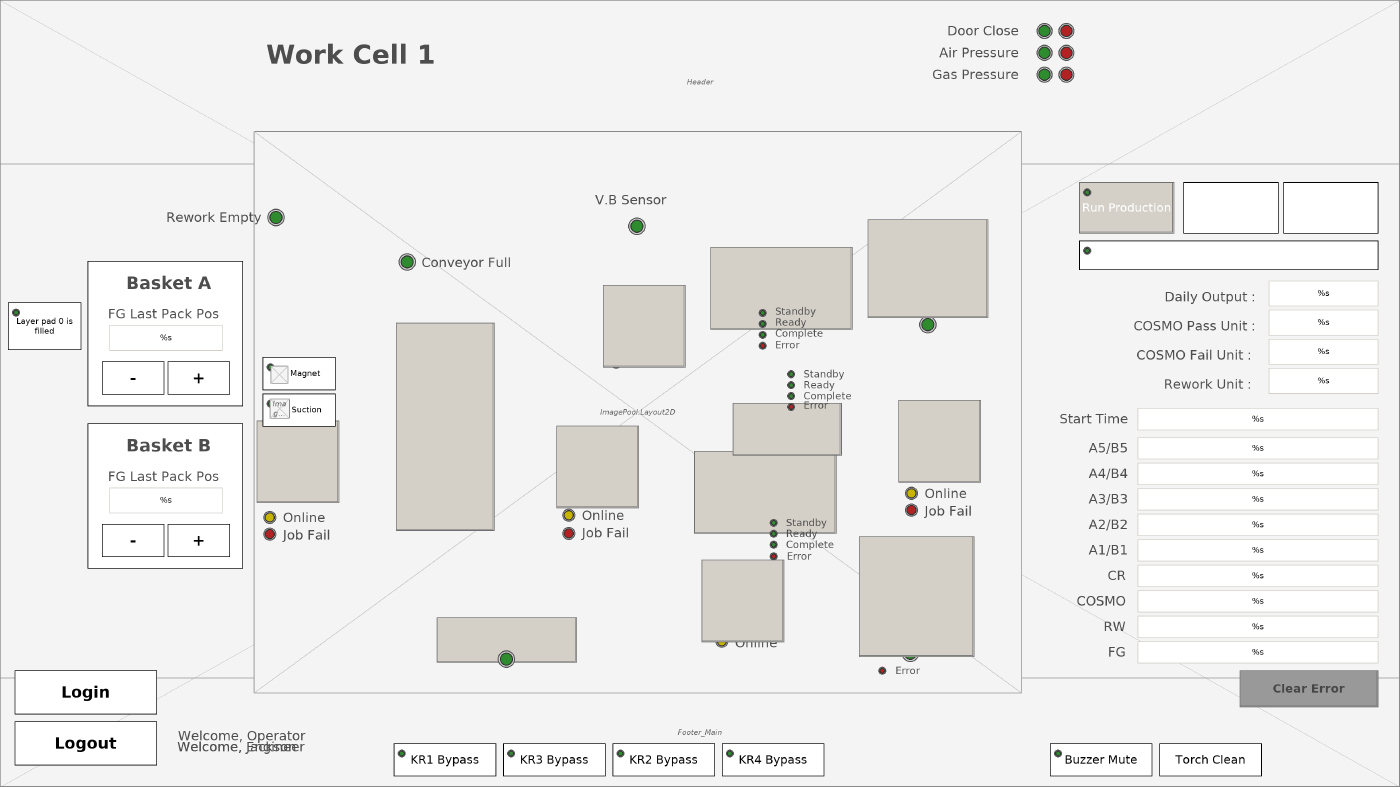
VISUALIZATION PAGE_MAIN  // 1920x1080
    Image (0,0 1920x1080), image: ImagePool.The-New-Silver-Backgrounds
    Frame (0,930 1920x150)
        shows Footer_Main()
        shows Footer_1()
    Frame (0,0 1920x225)
        shows Header()
    Label (362,45 650x60), "Work Cell 1"
    RoundedRectangle (1760,250 130x70), "Reset Production"
        OnMouseClick: OpenDialog Dialog=MSG_BOX_RESET, OpenModal=True, OpenCentered=True
    RoundedRectangle (20,990 195x60), "Logout"
        OnMouseClick: VisuUserMgmt Type=Logout
        OnMouseClick: execute {
            LOGFILE( sLogEvent	 := MSG.EVENT_BTN,
            		 sLogComp	 := MSG.COMP_HMI,
            		 sLogAction	 := MSG.ACTION_LOGOUT,
            	 	 logFlag	 := TRUE);
        }
    RoundedRectangle (20,920 195x60), "Login"
        tap MAIN.BTN_LOG
        OnMouseClick: VisuUserMgmt Type=Login
        OnMouseClick: execute {
            LOGFILE( sLogEvent	 := MSG.EVENT_BTN,
            		 sLogComp	 := MSG.COMP_HMI,
            		 sLogAction	 := MSG.ACTION_LOGIN,
            	 	 logFlag	 := TRUE);
        }
    Label (240,1005 200x40), "Welcome, Engineer"
    Label (240,1005 200x40), "Welcome, Jackson"
    Label (241,990 200x40), "Welcome, Operator"
    RoundedRectangle (120,358 213x199)
    Label (170,366 119x45), "Basket A"
    RoundedRectangle (140,496 85x45), "-"
        tap JIG.BasketA_Minus
        OnMouseClick: execute {
            LOGFILE( sLogEvent	 := MSG.EVENT_BTN,
            		 sLogComp	 := MSG.COMP_FG,
            		 sLogAction	 := MSG.ACTION_BSKTA_MINUS,
            	 	 logFlag	 := TRUE);
        }
    RoundedRectangle (230,496 85x45), "+"
        tap JIG.BasketA_Plus
        OnMouseClick: execute {
            LOGFILE( sLogEvent	 := MSG.EVENT_BTN,
            		 sLogComp	 := MSG.COMP_FG,
            		 sLogAction	 := MSG.ACTION_BSKTA_PLUS,
            	 	 logFlag	 := TRUE);
        }
    Textfield (150,446 155x35), "%s", text variable: GVL.Basket_A_Counter
    Label (145,416 173x30), "FG Last Pack Pos"
    RoundedRectangle (120,581 213x199)
    Label (170,589 119x45), "Basket B"
    RoundedRectangle (140,719 85x45), "-"
        tap JIG.BasketB_Minus
        OnMouseClick: execute {
            LOGFILE( sLogEvent	 := MSG.EVENT_BTN,
            		 sLogComp	 := MSG.COMP_FG,
            		 sLogAction	 := MSG.ACTION_BSKTA_MINUS,
            	 	 logFlag	 := TRUE);
        }
    RoundedRectangle (230,719 85x45), "+"
        tap JIG.BasketB_Plus
        OnMouseClick: execute {
            LOGFILE( sLogEvent	 := MSG.EVENT_BTN,
            		 sLogComp	 := MSG.COMP_FG,
            		 sLogAction	 := MSG.ACTION_BSKTB_PLUS,
            	 	 logFlag	 := TRUE);
        }
    Textfield (150,669 155x35), "%s", text variable: GVL.Basket_B_Counter
    Label (145,639 173x30), "FG Last Pack Pos"
    Image (348,180 1053x771), image: ImagePool.Layout2D
    Lamp1 (865,430 27x27), variable: KR3.bInBit[1,6], style: Lamp-Lamp1-Green
    Lamp1 (1010,815 27x27), variable: KR4.bInBit[1,6], style: Lamp-Lamp1-Green
    Lamp1 (1275,600 27x27), variable: KR5.bInBit[1,6], style: Lamp-Lamp1-Green
    Lamp1 (800,625 27x27), variable: KR2.bInBit[1,6], style: Lamp-Lamp1-Green
    Lamp1 (360,700 20x20), variable: KR1.KROnline, style: Lamp-Lamp1-Yellow
    Button (543,443 135x285)
        OnMouseClick: change screen: PAGE_CoolRack
        OnMouseClick: execute {
            LOGFILE( sLogEvent	 := MSG.EVENT_PAGE,
            		 sLogComp	 := MSG.COMP_CR,
            		 sLogAction	 := MSG.ACTION_COOLRACK,
            	 	 logFlag	 := TRUE);
        }
    Button (599,847 192x62)
        OnMouseClick: change screen: PAGE_COSMO
        OnMouseClick: execute {
            LOGFILE( sLogEvent	 := MSG.EVENT_PAGE,
            		 sLogComp	 := MSG.COMP_CM,
            		 sLogAction	 := MSG.ACTION_COSMO,
            	 	 logFlag	 := TRUE);
        }
    Lamp1 (681,891 27x27), variable: GVL.COSMO_Ready, style: Lamp-Lamp1-Green
    Lamp1 (860,297 27x27), variable: GVL.VibBowl_Ready, style: Lamp-Lamp1-Green
    Label (813,252 255x45), "V.B Sensor"
    Lamp1 (1259,432 27x27), variable: INFEED_RACK.IFRack_Ready, style: Lamp-Lamp1-Green
    Lamp1 (1235,883 27x27), variable: GVL.JIGC_Standby, style: Lamp-Lamp1-Green
    Button (1178,736 158x165)
        OnMouseClick: change screen: PAGE_TTorch
        OnMouseClick: execute {
            LOGFILE( sLogEvent	 := MSG.EVENT_PAGE,
            		 sLogComp	 := MSG.COMP_TT,
            		 sLogAction	 := MSG.ACTION_TT,
            	 	 logFlag	 := TRUE);
        }
    Button (974,339 195x113)
        OnMouseClick: change screen: PAGE_JIG_A
        OnMouseClick: execute {
            LOGFILE( sLogEvent	 := MSG.EVENT_PAGE,
            		 sLogComp	 := MSG.COMP_JIGA,
            		 sLogAction	 := MSG.ACTION_JIGA,
            	 	 logFlag	 := TRUE);
        }
    Button (952,619 195x113)
        OnMouseClick: change screen: PAGE_JIG_C
        OnMouseClick: execute {
            LOGFILE( sLogEvent	 := MSG.EVENT_PAGE,
            		 sLogComp	 := MSG.COMP_JIGC,
            		 sLogAction	 := MSG.ACTION_JIGC,
            	 	 logFlag	 := TRUE);
        }
    Button (1005,553 149x72)
        OnMouseClick: change screen: PAGE_JIG_B
        OnMouseClick: execute {
            LOGFILE( sLogEvent	 := MSG.EVENT_PAGE,
            		 sLogComp	 := MSG.COMP_JIGB,
            		 sLogAction	 := MSG.ACTION_JIGB,
            	 	 logFlag	 := TRUE);
        }
    Lamp1 (365,285 27x27), variable: GVL.Rework_Empty, style: Lamp-Lamp1-Green
    Lamp1 (545,346 27x27), variable: GVL.Conveyor_Full, style: Lamp-Lamp1-Green
    Label (225,276 146x45), "Rework Empty"
    Label (575,338 130x45), "Conveyor Full"
    Lamp1 (360,723 20x20), variable: KR1.bInBit[4,0], style: Lamp-Lamp1-Red
    Lamp1 (1240,690 20x20), variable: KR5.bInBit[4,7], style: Lamp-Lamp1-Red
    Lamp1 (770,722 20x20), variable: KR2.bInBit[3,4], style: Lamp-Lamp1-Red
    Lamp1 (395,633 27x27), variable: KR1.bInBit[1,6], style: Lamp-Lamp1-Green
    Label (385,722 80x25), "Job Fail"
    Label (385,698 80x25), "Online"
    Lamp1 (770,697 20x20), variable: KR2.KROnline, style: Lamp-Lamp1-Yellow
    Label (795,719 80x25), "Job Fail"
    Label (795,695 80x25), "Online"
    Lamp1 (1240,667 20x20), variable: KR5.KROnline, style: Lamp-Lamp1-Yellow
    Label (1265,689 80x25), "Job Fail"
    Label (1265,665 80x25), "Online"
    Lamp1 (835,487 20x20), variable: KR3.KROnline, style: Lamp-Lamp1-Yellow
    Label (860,485 80x25), "Online"
    Lamp1 (980,870 20x20), variable: KR4.KROnline, style: Lamp-Lamp1-Yellow
    Label (1005,870 80x25), "Online"
    Button (827,391 113x113)
        OnMouseClick: change screen: PAGE_KR3
        OnMouseClick: execute {
            LOGFILE( sLogEvent	 := MSG.EVENT_PAGE,
            		 sLogComp	 := MSG.COMP_KR3,
            		 sLogAction	 := MSG.ACTION_KR3,
            	 	 logFlag	 := TRUE);
        }
    Button (763,584 113x113)
        OnMouseClick: change screen: PAGE_KR2
        OnMouseClick: execute {
            LOGFILE( sLogEvent	 := MSG.EVENT_PAGE,
            		 sLogComp	 := MSG.COMP_KR2,
            		 sLogAction	 := MSG.ACTION_KR2,
            	 	 logFlag	 := TRUE);
        }
    Button (962,768 113x113)
        OnMouseClick: change screen: PAGE_KR4
        OnMouseClick: execute {
            LOGFILE( sLogEvent	 := MSG.EVENT_PAGE,
            		 sLogComp	 := MSG.COMP_KR4,
            		 sLogAction	 := MSG.ACTION_KR4,
            	 	 logFlag	 := TRUE);
        }
    Button (1232,549 113x113)
        OnMouseClick: change screen: PAGE_KR5
        OnMouseClick: execute {
            LOGFILE( sLogEvent	 := MSG.EVENT_PAGE,
            		 sLogComp	 := MSG.COMP_KR5,
            		 sLogAction	 := MSG.ACTION_KR5,
            	 	 logFlag	 := TRUE);
        }
    Button (352,577 113x113)
        OnMouseClick: change screen: PAGE_KR1_Tab
        OnMouseClick: execute {
            LOGFILE( sLogEvent	 := MSG.EVENT_PAGE,
            		 sLogComp	 := MSG.COMP_KR1,
            		 sLogAction	 := MSG.ACTION_KR1,
            	 	 logFlag	 := TRUE);
        }
    Label (1500,425 225x45), "COSMO Pass Unit :"
    Textfield (1740,425 150x35), "%s", text variable: GVL.Pass_Counter
    Textfield (1740,465 150x35), "%s", text variable: GVL.Fail_Counter
    Label (1500,465 225x45), "COSMO Fail Unit :"
    Textfield (1560,880 330x30), "%s", text variable: AUTO_MODE.processnameFG
    Group (1430,705 460x30)
        Textfield (130,0 330x30), "%s", text variable: AUTO_MODE.processnameA2
        Label (0,0 120x30), "A2/B2"
    Group (1430,740 460x30)
        Textfield (130,0 330x30), "%s", text variable: AUTO_MODE.processnameA1
        Label (0,0 120x30), "A1/B1"
    Textfield (1560,600 330x30), "%s", text variable: AUTO_MODE.processnameA5
    Label (1430,600 120x30), "A5/B5"
    Group (1430,635 460x30)
        Textfield (130,0 330x30), "%s", text variable: AUTO_MODE.processnameA4
        Label (0,0 120x30), "A4/B4"
    Group (1430,670 460x30)
        Textfield (130,0 330x30), "%s", text variable: AUTO_MODE.processnameA3
        Label (0,0 120x30), "A3/B3"
    Label (1472,880 75x30), "FG"
    Group (1472,845 418x30)
        Textfield (88,0 330x30), "%s", text variable: AUTO_MODE.processnameRW
        Label (0,0 75x30), "RW"
    Group (1472,775 418x30)
        Textfield (88,0 330x30), "%s", text variable: AUTO_MODE.processnameCR
        Label (0,0 75x30), "CR"
    Group (1455,810 435x30)
        Textfield (105,0 330x30), "%s", text variable: AUTO_MODE.processnameCOSMO
        Label (0,0 92x30), "COSMO"
    Lamp1 (1260,358 20x20), variable: INFEED_RACK.IFRack_Ready, style: Lamp-Lamp1-Yellow
    Button (1190,301 165x135)
        OnMouseClick: change screen: PAGE_InfeedRack
        OnMouseClick: execute {
            LOGFILE( sLogEvent	 := MSG.EVENT_PAGE,
            		 sLogComp	 := MSG.COMP_IR,
            		 sLogAction	 := MSG.ACTION_INFEEDRACK,
            	 	 logFlag	 := TRUE);
        }
    Label (1500,385 225x45), "Daily Output :"
    Textfield (1740,385 150x35), "%s", text variable: GVL.daily_output
    Label (1500,505 225x45), "Rework Unit :"
    Textfield (1740,505 150x35), "%s", text variable: GVL.Rework_Counter
    RoundedRectangle (1480,330 410x40), "Welding Mode"
        toggle SAFETY_SENSOR.WELDING_MODE
        OnMouseClick: execute {  }
    RoundedRectangle (1623,250 130x70), "Halt Production", input disabled if: MAIN.btnTorchClean
        OnMouseClick: execute {
            KR1.bOutBit[1,0]:= FALSE;
            KR2.bOutBit[1,0]:= FALSE;
            KR3.bOutBit[1,0]:= FALSE;
            KR4.bOutBit[1,0]:= FALSE;
            KR5.bOutBit[1,0]:= FALSE;
            LOGFILE( sLogEvent	 := MSG.EVENT_BTN,
            		 sLogComp	 := MSG.COMP_HMI,
            		 sLogAction	 := MSG.ACTION_STOP,
            	 	 logFlag	 := TRUE);
            AUTO_MODE.Halt_Production := TRUE;
            AUTO_MODE.AutoMode := False;
        }
    Button (1480,250 130x70), "Run Production", pressed state: AUTO_MODE.AutoMode, input disabled if: MAIN.btnTorchClean
        toggle AUTO_MODE.AutoMode
        OnMouseClick: execute {
            LOGFILE( sLogEvent	 := MSG.EVENT_BTN,
            		 sLogComp	 := MSG.COMP_HMI,
            		 sLogAction	 := MSG.ACTION_START,
            	 	 logFlag	 := TRUE);
            IF AUTO_MODE.AutoMode THEN
            	AUTO_MODE.Start_time := MAIN.fb_TimeStamp.SystemTime;
            END_IF
        }
    Lamp1 (1485,255 12x18), variable: AUTO_MODE.AutoMode, style: Lamp-Lamp1-Green
    Textfield (1560,560 330x30), "%s", text variable: AUTO_MODE.Start_time
    Label (1430,560 120x30), "Start Time"
    Lamp1 (1485,335 12x18), variable: SAFETY_SENSOR.WELDING_MODE, style: Lamp-Lamp1-Green
    Group (1250,20 225x105)
        Group (0,0 225x45)
            Label (0,0 150x45), "Door Close"
            Lamp1 (170,10 25x25), variable: SAFETY_SENSOR.SENSOR_SAFETY_DOOR_CLOSE, style: Lamp-Lamp1-Green
            Lamp1 (200,10 25x25), variable: not SAFETY_SENSOR.SENSOR_SAFETY_DOOR_CLOSE, style: Lamp-Lamp1-Red
        Label (0,30 150x45), "Air Pressure"
        Lamp1 (170,40 25x25), variable: SAFETY_SENSOR.SENSOR_AIR_PRESSURE_OK, style: Lamp-Lamp1-Green
        Lamp1 (200,40 25x25), variable: not SAFETY_SENSOR.SENSOR_AIR_PRESSURE_OK or SAFETY_SENSOR.SENSOR_AIR_PRESSURE_HIGH, style: Lamp-Lamp1-Red
        Label (0,60 150x45), "Gas Pressure"
        Lamp1 (170,70 25x25), variable: SAFETY_SENSOR.SENSOR_GAS_PRESSURE_OK, style: Lamp-Lamp1-Green
        Lamp1 (200,70 25x25), variable: not SAFETY_SENSOR.SENSOR_GAS_PRESSURE_OK or SAFETY_SENSOR.SENSOR_GAS_PRESSURE_HIGH, style: Lamp-Lamp1-Red
    Group (1079,506 100x45)
        Lamp1 (0,0 12x15), variable: GVL.JIGB_Standby, style: Lamp-Lamp1-Green
        Lamp1 (0,15 12x15), variable: GVL.JIGB_Ready, style: Lamp-Lamp1-Green
        Label (20,0 80x15), "Standby"
        Label (20,15 80x15), "Ready"
        Label (20,30 80x15), "Complete"
        Lamp1 (0,30 12x15), variable: GVL.JIGB_Complete, style: Lamp-Lamp1-Green
    Lamp1 (1040,422 12x15), variable: GVL.JIGA_Standby, style: Lamp-Lamp1-Green
    Lamp1 (1040,437 12x15), variable: GVL.JIGA_Ready, style: Lamp-Lamp1-Green
    Label (1060,420 80x15), "Standby"
    Label (1060,435 80x15), "Ready"
    Label (1060,450 80x15), "Complete"
    Lamp1 (1040,452 12x15), variable: GVL.JIGA_Complete, style: Lamp-Lamp1-Green
    Lamp1 (1055,710 12x15), variable: GVL.JIGC_Standby, style: Lamp-Lamp1-Green
    Lamp1 (1055,725 12x15), variable: GVL.JIGC_Ready, style: Lamp-Lamp1-Green
    Label (1075,710 80x15), "Standby"
    Label (1075,725 80x15), "Ready"
    Label (1075,740 80x15), "Complete"
    Lamp1 (1055,740 12x15), variable: GVL.JIGC_Complete, style: Lamp-Lamp1-Green
    Button (1700,920 190x50), "Clear Error", pressed state: MAIN.btn_Reset or MAIN.Reset_State
        toggle GVL.ClearError
        OnMouseClick: execute {
            LOGFILE( sLogEvent	 := MSG.EVENT_BTN,
            		 sLogComp	 := MSG.COMP_HMI,
            		 sLogAction	 := MSG.ACTION_CLEAR_ERROR,
            	 	 logFlag	 := TRUE);
        }
    Label (1060,466 80x15), "Error"
    Lamp1 (1040,467 12x15), variable: AUTO_MODE.JIGA_ErrorState, style: Lamp-Lamp1-Red
    Lamp1 (1079,551 12x15), variable: AUTO_MODE.JIGB_ErrorState, style: Lamp-Lamp1-Red
    Label (1099,549 80x15), "Error"
    Lamp1 (1055,756 12x15), variable: AUTO_MODE.JIGC_ErrorState, style: Lamp-Lamp1-Red
    Label (1076,756 80x15), "Error"
    Lamp1 (1204,913 12x15), variable: AUTO_MODE.TT_ErrorState, style: Lamp-Lamp1-Red
    Label (1225,913 80x15), "Error"
    RoundedRectangle (1590,1020 140x45), "Torch Clean"
        toggle MAIN.btnTorchClean
        OnMouseClick: execute {  }
    Group (1440,1020 140x45)
        RoundedRectangle (0,0 140x45), "Buzzer Mute"
            toggle TL.Buzzer_mute
            OnMouseClick: execute {  }
        Lamp1 (5,5 12x18), variable: TL.Buzzer_mute, style: Lamp-Lamp1-Green
    Group (840,1020 290x45)
        Group (150,0 140x45)
            RoundedRectangle (0,0 140x45), "KR4 Bypass"
                OnMouseClick: OpenDialog Dialog=MSG_KR4_BP, OpenModal=True, OpenCentered=True
            Lamp1 (5,5 12x18), variable: GVL.KR4_bypass, style: Lamp-Lamp1-Green
        RoundedRectangle (0,0 140x45), "KR2 Bypass"
            OnMouseClick: OpenDialog Dialog=MSG_KR2_BP, OpenModal=True, OpenCentered=True
        Lamp1 (5,5 12x18), variable: GVL.KR2_bypass, style: Lamp-Lamp1-Green
    RoundedRectangle (690,1020 140x45), "KR3 Bypass"
        OnMouseClick: OpenDialog Dialog=MSG_KR3_BP, OpenModal=True, OpenCentered=True
    Lamp1 (695,1025 12x18), variable: GVL.KR3_bypass, style: Lamp-Lamp1-Green
    RoundedRectangle (540,1020 140x45), "KR1 Bypass"
        OnMouseClick: OpenDialog Dialog=MSG_KR1_BP, OpenModal=True, OpenCentered=True
    Lamp1 (545,1025 12x18), variable: GVL.KR1_bypass, style: Lamp-Lamp1-Green
    Group (360,490 100x45)
        RoundedRectangle (0,0 100x45), "Magnet"
            OnMouseClick: OpenDialog Dialog=MSG_EOAT, OpenModal=True, OpenCentered=True
        Lamp1 (5,5 12x18), variable: GVL.KR1_EOAT_FILL, style: Lamp-Lamp1-Green
        Image (11,12 24x24), image: ImagePool.001-resources
    Group (360,540 100x45)
        RoundedRectangle (0,0 100x45), "Suction"
            OnMouseClick: OpenDialog Dialog=MSG_EOAT_SUCTION, OpenModal=True, OpenCentered=True
        Lamp1 (5,5 12x18), variable: GVL.KR1_EOAT_SUCTION, style: Lamp-Lamp1-Green
        Image (10,7 27x27), angle 180, image: ImagePool.002-plunger
    RoundedRectangle (11,415 100x65), "Layer pad 0 is filled"
        toggle GVL.LAYERPAD0
    Lamp1 (16,420 12x18), variable: GVL.LAYERPAD0, style: Lamp-Lamp1-Green
END_VISUALIZATION

(* stored: Version 1.1.0.1, ProductVersion 3.1.4024.12
   Visu PAGE_MAIN: Id {ca9ab701-d0c5-4665-b45c-c9c71481d4ca} *)
